FUNCTION_BLOCK InputLogger (* Extracted Composite Function Block Type *)
  (* Version 11/2/2016, chivdan *)
  PACKAGE Main;
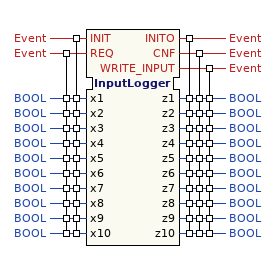
  EVENT_INPUT
    INIT WITH x1, x2, x3, x4, x5, x6, x7, x8, x9, x10; (* Initialization request *)
    REQ WITH x1, x2, x3, x4, x5, x6, x7, x8, x9, x10; (* Normal Execution Request *)
  END_EVENT
  EVENT_OUTPUT
    INITO WITH z1, z2, z3, z4, z5, z6, z7, z8, z9, z10; (* Initialization confirmation event *)
    CNF WITH z1, z2, z3, z4, z5, z6, z7, z8, z9, z10;
    WRITE_INPUT WITH z1, z2, z3, z4, z5, z6, z7, z8, z9, z10; (* Execution Confirmation *)
  END_EVENT
  VAR_INPUT
    x1 : BOOL; (* Argument *)
    x2 : BOOL; (* Argument *)
    x3 : BOOL; (* Argument *)
    x4 : BOOL; (* Argument *)
    x5 : BOOL; (* Argument *)
    x6 : BOOL; (* Argument *)
    x7 : BOOL; (* Argument *)
    x8 : BOOL; (* Argument *)
    x9 : BOOL; (* Argument *)
    x10 : BOOL; (* Argument *)
  END_VAR
  VAR_OUTPUT
    z1 : BOOL;
    z2 : BOOL;
    z3 : BOOL;
    z4 : BOOL;
    z5 : BOOL;
    z6 : BOOL;
    z7 : BOOL;
    z8 : BOOL;
    z9 : BOOL;
    z10 : BOOL;
  END_VAR
  FBS
    FB5 : ANY2ANY_-715679919; {SET_ATTRIBUTE(Configuration.GenericFBType.InterfaceParams, Runtime.Standard#CNT:=10;IN${CNT$}:BOOL,BOOL,BOOL,BOOL,BOOL,BOOL,BOOL,BOOL,BOOL,BOOL;OUT${CNT$}:INT,INT,INT,INT,INT,INT,INT,INT,INT,INT)}
    InputLogger : LOGGER_862393804(MESSAGE := in=REQ[${1}${2}${3}${4}${5}${6}${7}${8}${9}${10}], QI := TRUE, LEVEL := 1, DEST := 1); {SET_ATTRIBUTE(Configuration.GenericFBType.InterfaceParams, Runtime.System#CNT:=10)}
    FB6 : ChangeDetector;
    FB1 : E_MERGE;
  END_FBS
  EVENT_CONNECTIONS
    FB5.CNF TO FB6.REQ;
    FB6.CNF TO InputLogger.REQ;
    REQ TO FB5.REQ;
    InputLogger.INITO TO INITO;
    InputLogger.CNF TO FB1.EI1;
    FB6.SAME TO FB1.EI2;
    FB1.EO TO CNF;
    InputLogger.INITO TO FB5.REQ;
    INIT TO FB6.INIT;
    FB6.INITO TO InputLogger.INIT;
    FB6.CNF TO WRITE_INPUT;
  END_CONNECTIONS
  DATA_CONNECTIONS
    FB5.OUT1 TO FB6.x1;
    FB5.OUT2 TO FB6.x2;
    FB5.OUT3 TO FB6.x3;
    FB5.OUT4 TO FB6.x4;
    FB5.OUT5 TO FB6.x5;
    FB5.OUT6 TO FB6.x6;
    FB5.OUT7 TO FB6.x7;
    FB5.OUT8 TO FB6.x8;
    FB5.OUT9 TO FB6.x9;
    FB5.OUT10 TO FB6.x10;
    FB6.z1 TO InputLogger.PARAM1;
    FB6.z2 TO InputLogger.PARAM2;
    FB6.z3 TO InputLogger.PARAM3;
    FB6.z4 TO InputLogger.PARAM4;
    FB6.z5 TO InputLogger.PARAM5;
    FB6.z6 TO InputLogger.PARAM6;
    FB6.z7 TO InputLogger.PARAM7;
    FB6.z8 TO InputLogger.PARAM8;
    FB6.z9 TO InputLogger.PARAM9;
    FB6.z10 TO InputLogger.PARAM10;
    x1 TO FB5.IN1;
    x2 TO FB5.IN2;
    x3 TO FB5.IN3;
    x4 TO FB5.IN4;
    x5 TO FB5.IN5;
    x6 TO FB5.IN6;
    x7 TO FB5.IN7;
    x8 TO FB5.IN8;
    x9 TO FB5.IN9;
    x10 TO FB5.IN10;
    x1 TO z1;
    x2 TO z2;
    x3 TO z3;
    x4 TO z4;
    x5 TO z5;
    x6 TO z6;
    x7 TO z7;
    x8 TO z8;
    x9 TO z9;
    x10 TO z10;
  END_CONNECTIONS
END_FUNCTION_BLOCK
